(* IEC 61131-3 sources: plc_generation_empirical_study/datasets/task_bank_lean_runtime_v0_1/tasks/C04_R11_lean_composite/negative_control, 1 file *)

(* ---- NC1.st ---- *)
FUNCTION_BLOCK C04_R11_lean_composite
VAR_INPUT
    A_Signal : BOOL;
    A_Arm : BOOL;
    B_Info : BOOL;
    B_Warning : BOOL;
    B_Trip : BOOL;
    B_Emergency : BOOL;
    B_Suppress : BOOL;
    SubsystemBEnable : BOOL;
    CrossReset : BOOL;
END_VAR
VAR_OUTPUT
    A_Pulse : BOOL;
    A_Armed : BOOL;
    B_Active : BOOL;
    B_Level : INT;
    CrossReady : BOOL;
    CrossBlocked : BOOL;
END_VAR
VAR
    A_PrevSignal : BOOL := FALSE;
END_VAR

A_Pulse := A_Arm AND (NOT A_Signal) AND A_PrevSignal;
A_Armed := A_Arm;
A_PrevSignal := A_Signal;

IF CrossReset THEN
    CrossReady := FALSE;
ELSIF A_Pulse THEN
    CrossReady := TRUE;
END_IF;
CrossBlocked := FALSE;

IF SubsystemBEnable AND CrossReady THEN
    IF B_Emergency THEN
        B_Level := 4;
        B_Active := TRUE;
    ELSIF B_Suppress THEN
        B_Level := 0;
        B_Active := FALSE;
    ELSIF B_Trip THEN
        B_Level := 3;
        B_Active := TRUE;
    ELSIF B_Warning THEN
        B_Level := 2;
        B_Active := TRUE;
    ELSIF B_Info THEN
        B_Level := 1;
        B_Active := TRUE;
    ELSE
        B_Level := 0;
        B_Active := FALSE;
    END_IF;
ELSE
    B_Active := FALSE;
    B_Level := 0;
END_IF;

END_FUNCTION_BLOCK
